TYPE T_SimDtChn :
STRUCT
	stDecision: T_Decision;
	intJob: INT;
	strTimestamp: STRING(24);
	intDataState: INT;
	/// 0=undef, 1=SimDataPLCToLineDone, 2=SimDataLineToPLCInWork
	intInternalSimState: USINT;
END_STRUCT
END_TYPE

(* stored: Version 1.1.0.1, ProductVersion 3.1.0.23
   DUT T_SimDtChn: Id {0658eb28-9a3a-4f86-878a-a5f5d18c5a01} *)
